INTERFACE I_JobEventCreation EXTENDS __SYSTEM.IQueryInterface

PROPERTY job : I_Job
GET
END_GET
SET
END_SET
END_PROPERTY

PROPERTY title : T_MaxString
GET
END_GET
SET
END_SET
END_PROPERTY

END_INTERFACE

(* stored: Version 1.1.0.1, ProductVersion 3.1.4026.13
   Itf I_JobEventCreation: Id {ceea12a6-9e9c-4ed6-b610-0c7ba67cc010}
   Property job: Id {9cf427a5-a4be-41e8-a7bc-623984129431}
   Get Get: Id {729e7e51-b4af-4ad1-80be-9b5ad74660fb}
   Set Set: Id {ba8b64fd-da95-45c5-8c1e-c1cbb32b714d}
   Property title: Id {5372dc68-e45d-40fa-89ac-ccce6675f7d9}
   Get Get: Id {81a29a1c-2f23-42ca-a32d-a602d65dbc46}
   Set Set: Id {786c2ffb-0e01-47ab-be6b-9c9575544184} *)
